# EPICS substitutions: iocBoot/ioc13BNC505/asynRecord.substitutions
file "$(ASYN)/db/asynRecord.db"
{
pattern
{P              R         PORT     ADDR  OMAX IMAX}
{13LAE500:     serial1   serial1    0    256  256}
#{13LAE500:     serial2   serial2    0    256  256}
}
